INTERFACE I_LinkedListChangedEvent EXTENDS I_Event

PROPERTY PUBLIC TargetLinkedList : I_LinkedList
GET
END_GET
END_PROPERTY

END_INTERFACE

(* stored: Version 1.1.0.1, ProductVersion 3.1.4024.12
   Itf I_LinkedListChangedEvent: Id {c85c578b-7217-462a-95bd-f7ca34c5bef6}
   Property TargetLinkedList: Id {e2a01b88-797d-426a-be82-58b3bf9e0094}
   Get Get: Id {b8addeda-d410-4bd2-825d-2eca24e55d07} *)
